// TwinCAT 3 PLC project Untitled2
// ProgramVersion: 3.1.4022.2
// libraries:
//   Tc2_Standard, * (Beckhoff Automation GmbH)
//   Tc2_System, * (Beckhoff Automation GmbH)
//   Tc3_Module, * (Beckhoff Automation GmbH)
// project tree:
//   / PlcTask.TcTTO
//   POUs/ MAIN.TcPOU
// real-time tasks:
//   TASK PlcTask: cycle T#10ms, priority 20, ADS port 350
// I/O:
//   DEVICE Device 3 (EtherCAT), AmsNetId 192.168.1.6.4.1
//     Term 7 (EK1100) [EK1100 EtherCAT Coupler (2A E-Bus)]
//       Term 8 (EL2004) [EL2004 4Ch. Dig. Output 24V, 0.5A]
//       Term 9 (EL1904) [EL1904, 4 Ch. Safety Input 24V, TwinSAFE]
//         modules: Module 1 (FSOES)
//       Term 10 (EL2904) [EL2904, 4 Ch. Safety Output 24V, 0.5A, TwinSAFE]
//         modules: Module 1 (FSOES), Module 2 (DO)
//       Term 11 (EL6900) [EL6900, TwinSAFE PLC]
//       Term 13 (EL9011) [EL9011 End Terminal]
//     Box 12 (EL6692) [EL6692 EtherCAT Bridge terminal (Secondary)]
// variable links:
//   Device 3 (EtherCAT) <-> Device 3 (EtherCAT)/Box 12 (EL6692)
//     Term 7 (EK1100)/Term 11 (EL6900)/ConnectionInputs/Message_4 TxPDO <-> IO Outputs/Var 134
//     Term 7 (EK1100)/Term 11 (EL6900)/ConnectionOutputs/Message_4 RxPDO <-> IO Inputs/Var 160
//   Device 3 (EtherCAT) <-> Device 3 (EtherCAT)/Term 7 (EK1100)/Term 11 (EL6900)
//     Term 7 (EK1100)/Term 9 (EL1904)/Module 1 (FSOES)/TxPDO/FSOE <-> ConnectionOutputs/Message_5 RxPDO
//   Device 3 (EtherCAT) <-> Device 3 (EtherCAT)/Term 7 (EK1100)/Term 9 (EL1904)
//     Term 7 (EK1100)/Term 11 (EL6900)/ConnectionInputs/Message_5 TxPDO <-> Module 1 (FSOES)/RxPDO/FSOE
//   Untitled2/Untitled2 Instance <-> Device 3 (EtherCAT)/Term 7 (EK1100)/Term 11 (EL6900)
//     PlcTask Outputs/MAIN.mErrACK <-> StandardOutputs/Standard In Var 1
//     PlcTask Outputs/MAIN.mRun <-> StandardOutputs/Standard In Var 2

CONFIGURATION Untitled2
    RESOURCE PLC ON TwinCAT3
        TASK PlcTask(INTERVAL := T#5ms, PRIORITY := 20);
        PROGRAM MAIN WITH PlcTask : MAIN;
    END_RESOURCE
END_CONFIGURATION

// ---- POUs/MAIN.TcPOU
PROGRAM MAIN
VAR
	mErrACK AT %Q*	: BOOL;
	mRun AT %Q*		: BOOL;
END_VAR

mRun := True;

END_PROGRAM
